(* IEC 61131-3 sources: OpenPLC_Tutorials/Ladder Logic and Ladder Diagram/02 NO and NC/02 NO and NC/build, 2 files *)

(* ---- plc.st ---- *)
TYPE
  LOGLEVEL : (CRITICAL, WARNING, INFO, DEBUG) := INFO;
END_TYPE

FUNCTION_BLOCK LOGGER
  VAR_INPUT
    TRIG : BOOL;
    MSG : STRING;
    LEVEL : LOGLEVEL := INFO;
  END_VAR
  VAR
    TRIG0 : BOOL;
  END_VAR

  IF TRIG AND NOT TRIG0 THEN
  {{
   LogMessage(GetFbVar(LEVEL),(char*)GetFbVar(MSG, .body),GetFbVar(MSG, .len));
  }}
  END_IF;
  TRIG0:=TRIG;
END_FUNCTION_BLOCK

PROGRAM NO_NC
  VAR
    NO_Contact : BOOL;
    NC_Contact : BOOL;
    Coil_1 : BOOL;
    Coil_2 : BOOL;
  END_VAR

  Coil_1 := NO_Contact;
  Coil_2 := NOT(NC_Contact);
END_PROGRAM

CONFIGURATION Config0

  RESOURCE Res0 ON PLC
    TASK task0(INTERVAL := T#20ms,PRIORITY := 0);
    PROGRAM instance0 WITH task0 : NO_NC;
  END_RESOURCE
END_CONFIGURATION

(* ---- generated_plc.st ---- *)
PROGRAM NO_NC
  VAR
    NO_Contact : BOOL;
    NC_Contact : BOOL;
    Coil_1 : BOOL;
    Coil_2 : BOOL;
  END_VAR

  Coil_1 := NO_Contact;
  Coil_2 := NOT(NC_Contact);
END_PROGRAM

CONFIGURATION Config0

  RESOURCE Res0 ON PLC
    TASK task0(INTERVAL := T#20ms,PRIORITY := 0);
    PROGRAM instance0 WITH task0 : NO_NC;
  END_RESOURCE
END_CONFIGURATION
